// Mitsubishi GX Works2 project: 단속동작   PLC: Q02/Q02H

PROGRAM MAIN
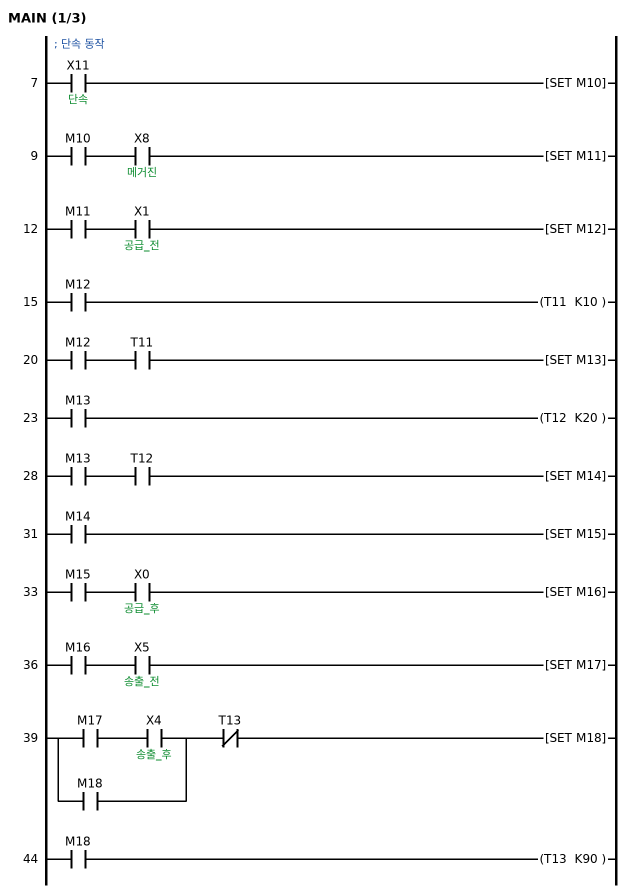
; 단속 동작
7     LD      X11  ; 단속
      SET     M10
9     LD      M10
      AND     X8  ; 메거진
      SET     M11
12    LD      M11
      AND     X1  ; 공급_전
      SET     M12
15    LD      M12
      OUT     T11 K10
20    LD      M12
      AND     T11
      SET     M13
23    LD      M13
      OUT     T12 K20
28    LD      M13
      AND     T12
      SET     M14
31    LD      M14
      SET     M15
33    LD      M15
      AND     X0  ; 공급_후
      SET     M16
36    LD      M16
      AND     X5  ; 송출_전
      SET     M17
39    LD      M17
      AND     X4  ; 송출_후
      OR      M18
      ANI     T13
      SET     M18
44    LD      M18
      OUT     T13 K90
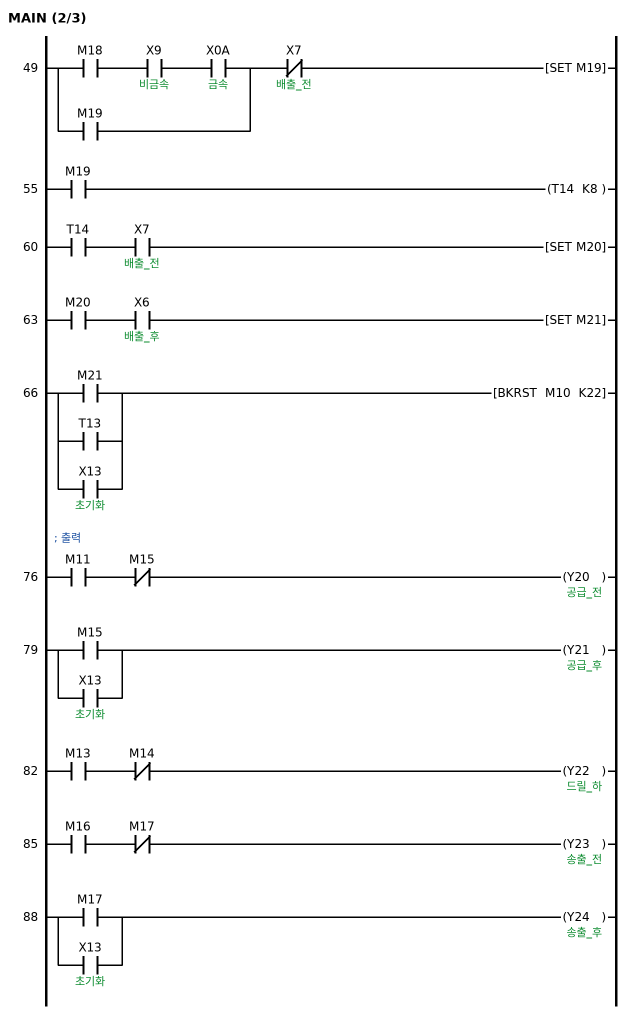
49    LD      M18
      AND     X9  ; 비금속
      AND     X0A  ; 금속
      OR      M19
      ANI     X7  ; 배출_전
      SET     M19
55    LD      M19
      OUT     T14 K8
60    LD      T14
      AND     X7  ; 배출_전
      SET     M20
63    LD      M20
      AND     X6  ; 배출_후
      SET     M21
66    LD      M21
      OR      T13
      OR      X13  ; 초기화
      BKRST   M10 K22
; 출력
76    LD      M11
      ANI     M15
      OUT     Y20  ; 공급_전
79    LD      M15
      OR      X13  ; 초기화
      OUT     Y21  ; 공급_후
82    LD      M13
      ANI     M14
      OUT     Y22  ; 드릴_하
85    LD      M16
      ANI     M17
      OUT     Y23  ; 송출_전
88    LD      M17
      OR      X13  ; 초기화
      OUT     Y24  ; 송출_후
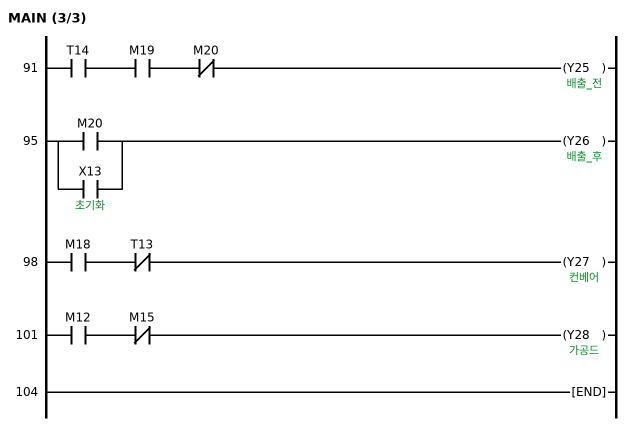
91    LD      T14
      AND     M19
      ANI     M20
      OUT     Y25  ; 배출_전
95    LD      M20
      OR      X13  ; 초기화
      OUT     Y26  ; 배출_후
98    LD      M18
      ANI     T13
      OUT     Y27  ; 컨베어
101   LD      M12
      ANI     M15
      OUT     Y28  ; 가공드
104   END
END_PROGRAM

// device comments not shown above
X2  ; 드릴_상
X3  ; 드릴_하
X10  ; 테스트
X12  ; 연속
Y29  ; 적색
Y2A  ; 황색
Y2B  ; 녹색
